	    REGION Niveaumessung
	        // Füllstand Versorgung Frischsäure
	        "Analogwert"(Deaktiviert:=FALSE,
	                                                                                                                                                                                                                                                                                                                                                                                                                                                                                                                                                                                                                                                                                                                                                                                                                                                                                                                                                                                                                                                                                                                                                                                                                                                                                                                                                                                                                                                                                                                                                                                                                                                                                                                                                                                                                                                                                                                                                                                                                                                                                                                                                                                                                                                                                                                                                                                                                                                                                                                                                                                                                                                                                                                                                                                                                                                                                                                                                                                                                                                                                                                                                                                                                                                                                                                                                                                                                                                                                                                                                                                                                                                                                                                                                                                                                                                                                                                                                                                                                                                                                                                                                                                                                                                                                                                                                                                                                                                                                                                                                                                                                                                                                                                                                                                                                                                                                                                                                                                                                                                                                                                                                                                                                                                                                                                                                                                                                                                                                                                                                                                                                                                                                                                                                                                                                                                                                                                                                                                                                                                                                                                                                                                                                                                                                                                                                                                                                                                                                                                                                                                                                                                                                                                                                                                                                                                                                                                                                                                                                                                                                                                                                                                                                                                                                                                                                                                                                                                                                                                                                                                                                                                                                                                                                                                                                                                                                                                                                                                                                                                                                                                                                                                                                                                                                                                                                                                                                                                                                                                                                                                                                                                                                                                                                                                                                                                                                                                                                                                                                                                                                                                                                                                                                                                                                                                                                                                                                                                                                                                                                                                                                                                                                                                                                                                                                                                                                                                                                                                                                                                                                                                                                                                                                                                                                                                                                                                                                                                                                                                                                                                                                                                                                                                                                                                                                                                                                                                                                                                                                                                                                                                                                                                                                                                                                                                                                                                                                                                                                                                                                                                                                                                                                                                                                                                                                                                                                                                                                                                                                                                                                                                                                                                                                                                                                                                                                                                                                                                                                                                                                                                                                                                                                                                                                                                                                                                                                                                                                                                                                                                                                                                                                                                                                                                                                                                                                                                                                                                                                                                                                                                                                                                                                                                                                                                                                                                                                                                                                                                                                                                                                                                                                                                                                                                                                                                                                                                                                                                                                                                                                                                                                                                                                                                                                                                                                                                                                                                                                                                                                                                                                                                                                                                                                                                                                                                                                                                                                                                                                                                                                                                                                                                                                                                                                                                                                                                                                                                                                                                                                                                                                                                                                                                                                                                                                                                                                                                                                                                                                                                                                                                                                                                                                                                                                                                                                                                                                                                                                                                                                                                                                                                                                                                                                                                                                                                                                                                                                                                                                                                                                                                                                                                                                                                                                                                                                                                                                                                                                                                                                                                                                                                                                                                                                                                                                                                                                                                                                                                                                                                                                                                                                                                                                                                                                                                                                                                                                                                                                                                                                                                                                                                                                                                                                                                                                                                                                                                                                                                                                                                                                                                                                                                                                                                                                                                                                                                                                                                                                                                                                                                                                                                                                                                                                                                                                                                                                                                                                                                                                                                                                                                                                                                                                                                                                                                                                                                                                                                                                                                                                                                                                                                                                                                                                                                                                                                                                                                                                                                                                                                                                                                                                                                                                                                                                                                                                                                                                                                                                                                                                                                                                                                                                                                                                                                                                                                                                                                                                                                                                                                                                                                                                                                                                                                                                                                                                                                                                                                                                                                                                                                                                                                                                                                                                                                                                                                                                                                                                                                                                                                                                                                                                                                                                                                                                                                                                                                                                                                                                                                                                                                                                                                                                                                                                                                                                                                                                                                                                                                                                                                                                                                                                                                                                                                                                                                                                                                                                                                                                                                                                                                                                                                                                                                                                                                                                                                                                                                                                                                                                                                                                                                                                                                                                                                                                                                                                                                                                                                                                                                                                                                                                                                                                                                                                                                                                                                                                                                                                                                                                                                                                                                                                                                                                                                                                                                                                                                                                                                                                                                                                                                                                                                                                                                                                                                                                                                                                                                                                                                                                                                                                                                                                                                                                                                                                                                                                                                                                                                                                                                                                                                                                                                                                                                                                                                                                                                                                                                                                                                                                                                                                                                                                                                                                                                                                                                                                                                                                                                                                                                                                                                                                                                                                                                                                                                                                                                                                                                                                                                                                                                                                                                                                                                                                                                                                                                                                                                                                                                                                                                                                                                                                                                                                                                                                                                                                                                                                                                                                                                                                                                                                                                                                                                                                                                                                                                                                                                                                                                                                                                                                                                                                                                                                                                                                                                                                                                                                                                                                                                                                                                                                                                                                                                                                                                                                                                                                                                                                                                                                                                                                                                                                                                                                                                                                                                                                                                                                                                                                                                                                                                                                                                                                                                                                                                                                                                                                                                                                                                                                                                                                                                                                                                                                                                                                                                                                                                                                                                                                                                                                                                                                                                                                                                                                                                                                                                                                                                                                                                                                                                                                                                                                                                                                                                                                                                                                                                                                                                                                                                                                                                                                                                                                                                                                                                                                                                                                                                                                                                                                                                                                                                                                                                                                                                                                                                                                                                                                                                                                                                                                                                                                                                                                                                                                                                                                                                                                                                                                                                                                                                                                                                                                                                                                                                                                                                                                                                                                                                                                                                                                                                                                                                                                                                                                                                                                                                                                                                                                                                                                                                                                                                                                                                                                                                                                                                                                                                                                                                                                                                                                                                                                                                                                                                                                                                                                                                                                                                                                                                                                                                                                                                                                                                                                                                                                                                                                                                                                                                                                                                                                                                                                                                                                                                                                                                                                                                                                                                                                                                                                                                                                                                                                                                                                                                                                                                                                                                                                                                                                                                                                                                                                                                                                                                                                                                                                                                                                                                                                                                                                                                                                                                                                                                                                                                                                                                                                                                                                                                                                                                                                                                                                                                                                                                                                                                                                                                                                                                                                                                                                                                                                                                                                                                                                                                                                                                                                                                                                                                                                                                                                                                                                                                                                                                                                                                                                                                                                                                                                                                                                                                                                                                                                                                                                                                                                                                                                                                                                                                                                                                                                                                                                                                                                                                                                                                                                                                                                                                                                                                                                                                                                                                                                                                                                                                                                                                                                                                                                                                                                                                                                                                                                                                                                                                                                                                                                                                                                                                                                                                                                                                                                                                                                                                                                                                                                                                                                                                                                                                                                                                                                                                                                                                                                                                                                                                                                                                                                                                                                                                                                                                                                                                                                                                                                                                                                                                                                                                                                                                                                                                                                                                                                                                                                                                                                                                                                                                                                                                                                                                                                                                                                                                                                                                                                                                                                                                                                                                                                                                                                                                                                                                                                                                                                                                                                                                                                                                                                                                                                                                                                                                                                                                                                                                                                                                                                                                                                                                                                                                                                                                                                                                                                                                                                                                                                                                                                                                                                                                                                                                                                                                                                                                                                                                                                                                                                                                                                                                                                                                                                                                                                                                                                                                                                                                                                                                                                                                                                                                                                                                                                                                                                                                                                                                                                                                                                                                                                                                                                                                                                                                                                                                                                                                                                                                                                                                                                                                                                                                                                                                                                                                                                                                                                                                                                                                                                                                                                                                                                                                                                                                                                                                                                                                                                                                                                                                                                                                                                                                                                                                                                                                                                                                                                                                                                                                                                                                                                                                                                                                                                                                                                                                                                                                                                                                                                                                                                                                                                                                                                                                                                                                                                                                                                                                                                                                                                                                                                                                                                                                                                                                                                                                                                                                                                                                                                                                                                                                                                                                                                                                                                                                                                                                                                                                                                                                                                                                                                                                                                                                                                                                                                                                                                                                                                                                                                                                                                                                                                                                                                                                                                                                                                                                                                                                                                                                                                                                                                                                                                                                                                                                                                                                                                                                                                                                                                                                                                                                                                                                                                                                                                                                                                                                                                                                                                                                                                                                                                                                                                                                                                                                                                                                                                                                                                                                                                                                                                                                                                                                                                                                                                                                                                                                                                                                                                                                                                                                                                                                                                                                                                                                                                                                                                                                                                                                                                                                                                                                                                                                                                                                                                                                                                                                                                                                                                                                                                                                                                                                                                                                                                                                                                                                                                                                                                                                                                                                                                                                                                                                                                                                                                                                                                                                                                                                                                                                                                                                                                                                                                                                                                                                                                                                                                                                                                                                                                                                                                                                                                                                                                                                                                                                                                                                                                                                                                                                                                                                                                                                                                                                                                                                                                                                                                                                                                                                                                                                                                                                                                                                                                                                                                                                                                                                                                                                                                                                                                                                                                                                                                                                                                                                                                                                                                                                                                                                                                                                                                                                                                                                                                                                                                                                                                                                                                                                                                                                                                                                                                                                                                                                                                                                                                                                                                                                                                                                                                                                                                                                                                                                                                                                                                                                                                                                                                                                                                                                                                                                                                                                                                                                                                                                                                                                                                                                                                                                                                                                                                                                                                                                                                                                                                                                                                                                                                                                                                                                                                                                                                                                                                                                                                                                                                                                                                                                                                                                                                                                                                                                                                                                                                                                                                                                                                                                                                                                                                                                                                                                                                                                                                                                                                                                                                                                                                                                                                                                                                                                                                                                                                                                                                                                                                                                                                                                                                                                                                                                                                                                                                                                                                                                                                                                                                                                                                                                                                                                                                                                                                                                                                                                                                                                                                                                                                                                                                                                                                                                                                                                                                                                                                                                                                                                                                                                                                                                                                                                                                                                                                                                                                                                                                                                                                                                                                                                                                                                                                                                                                                                                                                                                                                                                                                                                                                                                                                                                                                                                                                                                                                                                                                                                                                                                                                                                                                                                                      EW := "EW_Niv_GP01.BL30",
	                     Messbereich_Min := "Analogwerte"."Niv_GP01.BL30".MB_min,
	                     Messbereich_Max := "Analogwerte"."Niv_GP01.BL30".MB_max,
	                     UG_Alarm := "Analogwerte"."Niv_GP01.BL30".UG_Alarm,
	                     OG_Alarm := "Analogwerte"."Niv_GP01.BL30".OG_Alarm,
	                     GF := "Analogwerte"."Niv_GP01.BL30".GF,
	                     Al_Drahtbruch => "Analogwerte"."Niv_GP01.BL30".Drahtbruch,
	                     Al_MW_ausserhalb => "Analogwerte"."Niv_GP01.BL30".ungueltig,
	                     Messwert := "Panel".IW."Niv_GP01.BL30");
	        // Füllstand Entsorgung Altsäure
	        "Analogwert"(Deaktiviert:=FALSE,
	                        EW := "EW_Niv_GP02.BL31",
	                     Messbereich_Min := "Analogwerte"."Niv_GP02.BL31".MB_min,
	                     Messbereich_Max := "Analogwerte"."Niv_GP02.BL31".MB_max,
	                     UG_Alarm := "Analogwerte"."Niv_GP02.BL31".UG_Alarm,
	                     OG_Alarm := "Analogwerte"."Niv_GP02.BL31".OG_Alarm,
	                     GF := "Analogwerte"."Niv_GP02.BL31".GF,
	                     Al_Drahtbruch => "Analogwerte"."Niv_GP02.BL31".Drahtbruch,
	                     Al_MW_ausserhalb => "Analogwerte"."Niv_GP02.BL31".ungueltig,
	                     Messwert := "Panel".IW."Niv_GP02.BL31");
	     END_REGION
	// pH-Messung
	     "Analogwert"(Deaktiviert:=FALSE,
	             EW := "EW_LW_BE",
	             Messbereich_Min := "Analogwerte".pH_WR01.MB_min,
	             Messbereich_Max := "Analogwerte".pH_WR01.MB_max,
	             UG_Alarm := "Analogwerte".pH_WR01.UG_Alarm,
	             OG_Alarm := "Analogwerte".pH_WR01.OG_Alarm,
	             GF := "Analogwerte".pH_WR01.GF,
	             Al_Drahtbruch => "Analogwerte".pH_WR01.Drahtbruch,
	             Al_MW_ausserhalb => "Analogwerte".pH_WR01.ungueltig,
	             Messwert := "Panel".IW."pH_BE");
	END_IF;
	
	REGION Manipulator
	    IF "Imp_10Hz" THEN // 8x Wägezelle, 2x Last
	        "Analogwert"(Deaktiviert:=FALSE,
	                     EW := "EW_WZ_links_1",
	                     Messbereich_Min := "Analogwerte".WZ_1_1.MB_min,
	                     Messbereich_Max := "Analogwerte".WZ_1_1.MB_max,
	                     UG_Alarm := "Analogwerte".WZ_1_1.UG_Alarm,
	                     OG_Alarm := "Analogwerte".WZ_1_1.OG_Alarm,
	                     GF := "Analogwerte".WZ_1_1.GF,
	                     Al_Drahtbruch => "Analogwerte".WZ_1_1.Drahtbruch,
	                     Al_MW_ausserhalb => "Analogwerte".WZ_1_1.ungueltig,
	                     Messwert := "DI_FW_1".HELP.WZ_links_1);
	        
	        "Analogwert"(Deaktiviert:=FALSE,
	                     EW := "EW_WZ_links_2",
	                     Messbereich_Min := "Analogwerte".WZ_1_2.MB_min,
	                     Messbereich_Max := "Analogwerte".WZ_1_2.MB_max,
	                     UG_Alarm := "Analogwerte".WZ_1_2.UG_Alarm,
	                     OG_Alarm := "Analogwerte".WZ_1_2.OG_Alarm,
	                     GF := "Analogwerte".WZ_1_2.GF,
	                     Al_Drahtbruch => "Analogwerte".WZ_1_2.Drahtbruch,
	                     Al_MW_ausserhalb => "Analogwerte".WZ_1_2.ungueltig,
	                     Messwert := "DI_FW_1".HELP.WZ_links_2);
	        
	        "Analogwert"(Deaktiviert:=FALSE,
	                     EW := "EW_WZ_links_3",
	                     Messbereich_Min := "Analogwerte".WZ_1_3.MB_min,
	                     Messbereich_Max := "Analogwerte".WZ_1_3.MB_max,
	                     UG_Alarm := "Analogwerte".WZ_1_3.UG_Alarm,
	                     OG_Alarm := "Analogwerte".WZ_1_3.OG_Alarm,
	                     GF := "Analogwerte".WZ_1_3.GF,
	                     Al_Drahtbruch => "Analogwerte".WZ_1_3.Drahtbruch,
	                     Al_MW_ausserhalb => "Analogwerte".WZ_1_3.ungueltig,
	                     Messwert := "DI_FW_1".HELP.WZ_links_3);
	        
	        "Analogwert"(Deaktiviert:=FALSE,
	                    EW := "EW_WZ_links_4",
	                     Messbereich_Min := "Analogwerte".WZ_1_4.MB_min,
	                     Messbereich_Max := "Analogwerte".WZ_1_4.MB_max,
	                     UG_Alarm := "Analogwerte".WZ_1_4.UG_Alarm,
	                     OG_Alarm := "Analogwerte".WZ_1_4.OG_Alarm,
	                     GF := "Analogwerte".WZ_1_4.GF,
	                     Al_Drahtbruch => "Analogwerte".WZ_1_4.Drahtbruch,
	                     Al_MW_ausserhalb => "Analogwerte".WZ_1_4.ungueltig,
	                     Messwert := "DI_FW_1".HELP.WZ_links_4);
	        
	        "Analogwert"(Deaktiviert:=FALSE,
	                     EW := "EW_WZ_rechts_1",
	                     Messbereich_Min := "Analogwerte".WZ_2_1.MB_min,
	                     Messbereich_Max := "Analogwerte".WZ_2_1.MB_max,
	                     UG_Alarm := "Analogwerte".WZ_2_1.UG_Alarm,
	                     OG_Alarm := "Analogwerte".WZ_2_1.OG_Alarm,
	                     GF := "Analogwerte".WZ_2_1.GF,
	                     Al_Drahtbruch => "Analogwerte".WZ_2_1.Drahtbruch,
	                     Al_MW_ausserhalb => "Analogwerte".WZ_2_1.ungueltig,
	                     Messwert := "DI_FW_1".HELP.WZ_rechts_1);
	        
	        "Analogwert"(Deaktiviert := FALSE,
	                     EW := "EW_WZ_rechts_2",
	                     Messbereich_Min := "Analogwerte".WZ_2_2.MB_min,
	                     Messbereich_Max := "Analogwerte".WZ_2_2.MB_max,
	                     UG_Alarm := "Analogwerte".WZ_2_2.UG_Alarm,
	                     OG_Alarm := "Analogwerte".WZ_2_2.OG_Alarm,
	                     GF := "Analogwerte".WZ_2_2.GF,
	                     Al_Drahtbruch => "Analogwerte".WZ_2_2.Drahtbruch,
	                     Al_MW_ausserhalb => "Analogwerte".WZ_2_2.ungueltig,
	                     Messwert := "DI_FW_1".HELP.WZ_rechts_2);
	        
	        "Analogwert"(Deaktiviert := FALSE,
	                     EW := "EW_WZ_rechts_3",
	                     Messbereich_Min := "Analogwerte".WZ_2_3.MB_min,
	                     Messbereich_Max := "Analogwerte".WZ_2_3.MB_max,
	                     UG_Alarm := "Analogwerte".WZ_2_3.UG_Alarm,
	                     OG_Alarm := "Analogwerte".WZ_2_3.OG_Alarm,
	                     GF := "Analogwerte".WZ_2_3.GF,
	                     Al_Drahtbruch => "Analogwerte".WZ_2_3.Drahtbruch,
	                     Al_MW_ausserhalb => "Analogwerte".WZ_2_3.ungueltig,
	                     Messwert := "DI_FW_1".HELP.WZ_rechts_3);
	        
	        "Analogwert"(Deaktiviert := FALSE,
	                     EW := "EW_WZ_rechts_4",
	                     Messbereich_Min := "Analogwerte".WZ_2_4.MB_min,
	                     Messbereich_Max := "Analogwerte".WZ_2_4.MB_max,
	                     UG_Alarm := "Analogwerte".WZ_2_4.UG_Alarm,
	                     OG_Alarm := "Analogwerte".WZ_2_4.OG_Alarm,
	                     GF := "Analogwerte".WZ_2_4.GF,
	                     Al_Drahtbruch => "Analogwerte".WZ_2_4.Drahtbruch,
	                     Al_MW_ausserhalb => "Analogwerte".WZ_2_4.ungueltig,
	                     Messwert := "DI_FW_1".HELP.WZ_rechts_4);
	        
	        "Analogwert"(Deaktiviert := FALSE,
	                     EW := "EW_Last_links",
	                     Messbereich_Min := "Analogwerte".Last_1.MB_min,
	                     Messbereich_Max := "Analogwerte".Last_1.MB_max,
	                     UG_Alarm := "Analogwerte".Last_1.UG_Alarm,
	                     OG_Alarm := "Analogwerte".Last_1.OG_Alarm,
	                     GF := "Analogwerte".Last_1.GF,
	                     Al_Drahtbruch => "Analogwerte".Last_1.Drahtbruch,
	                     Al_MW_ausserhalb => "Analogwerte".Last_1.ungueltig,
	                     Messwert := "DI_FW_1".HELP.Last_1);
	        
	        "Analogwert"(Deaktiviert:=FALSE,
	                     EW := "EW_Last_rechts",
	                     Messbereich_Min := "Analogwerte".Last_2.MB_min,
	                     Messbereich_Max := "Analogwerte".Last_2.MB_max,
	                     UG_Alarm := "Analogwerte".Last_2.UG_Alarm,
	                     OG_Alarm := "Analogwerte".Last_2.OG_Alarm,
	                     GF := "Analogwerte".Last_2.GF,
	                     Al_Drahtbruch => "Analogwerte".Last_2.Drahtbruch,
	                     Al_MW_ausserhalb => "Analogwerte".Last_2.ungueltig,
	                     Messwert := "DI_FW_1".HELP.Last_2);
	    END_IF;
	
	END_REGION
	
END_FUNCTION

FUNCTION "Analogwert" : Void
{ S7_Optimized_Access := 'TRUE' }
VERSION : 0.1
   VAR_INPUT 
      Deaktiviert : Bool;
      EW : Int;
      Messbereich_Min : Real;
      Messbereich_Max : Real;
      UG_Alarm : Real;
      OG_Alarm : Real;
      GF : Real;
   END_VAR

   VAR_OUTPUT 
      Al_Drahtbruch : Bool;
      Al_MW_ausserhalb : Bool;
   END_VAR

   VAR_IN_OUT 
      Messwert : Real;
   END_VAR

   VAR_TEMP 
      akt_Messwert : Real;
      Messbereich : Real;
      Eingangswert : Real;
   END_VAR

   VAR CONSTANT 
      Drahtbruchkennung : Int := 16#7FFF;
      Defekt : Int := 16#8000;
      EW_min : Real;
      EW_max : Real := 27648.0;   // SIEMENS-Baugruppe (0x6C00)
   END_VAR


BEGIN
	IF #Deaktiviert THEN //20.01.22
	    #Al_Drahtbruch := FALSE;
	    #Al_MW_ausserhalb := false;
	    #Messwert := 0.0;
	    
	ELSIF (#EW = #Drahtbruchkennung) OR (#EW = #Defekt) THEN
	    #Al_Drahtbruch := TRUE;
	    #Al_MW_ausserhalb := false;
	    #Messwert := 0.0;
	ELSE
	    #Al_Drahtbruch := FALSE;
	    #Messbereich := (#EW_max - #EW_min);
	    #Eingangswert := DINT_TO_REAL(INT_TO_DINT(#EW));
	    
	    #akt_Messwert := ((#Eingangswert - #EW_min) * #Messbereich_Max / #Messbereich) + ((#EW_max - #Eingangswert) * #Messbereich_Min / #Messbereich);
	      
	    IF (#GF <= 0.0) OR #GF >= 1.0 THEN
	        #Messwert := #akt_Messwert;
	    ELSE
	         #Messwert := (#akt_Messwert * #GF) + ((1.0 - #GF) * #Messwert);
	     END_IF;
	     #Al_MW_ausserhalb := (#Messwert < #UG_Alarm) OR (#Messwert > #OG_Alarm);
	    
	END_IF;
	
END_FUNCTION

FUNCTION "BA_WXL" : Void   // FC4, STL
{ S7_Optimized_Access := 'FALSE' }
AUTHOR : MS
// stored: AutoNumber false
   VAR_TEMP
      Evnt_Nbr : Byte;
   END_VAR
   VAR CONSTANT
      Not_Halt : USInt;
      Tipp : USInt := 1;
      Hand : USInt := 2;
      Automat_Aus : USInt := 3;
      Automat_Ein : USInt := 4;
   END_VAR
BEGIN

NETWORK
TITLE = Not-Aus ist betätigt
      A     "DB_ANLAGE".config.Anl_getaktet;
      =     "DB_Panel_OVERVIEW".SPS_getaktet;

      A     "DB_ANLAGE".IN.S_Not_Aus;
      JC    off;

//Automatikbetrieb
      A     "DB_ANLAGE".BA.Not_Aus;
      R     "DB_ANLAGE".BA.Not_Aus;
      R     "DB_ANLAGE".BA.Tippbetrieb;
      R     "DB_ANLAGE".BA.Handbetrieb;
      R     "DB_ANLAGE".BA.Automat_ein;
      S     "DB_ANLAGE".BA.Automat_aus;

      A     "DB_ANLAGE".IN.Automat_ein;
      FP    "DB_ANLAGE".BA.FP_Automat_ein;
      R     "DB_ANLAGE".BA.Not_Aus;
      R     "DB_ANLAGE".BA.Tippbetrieb;
      R     "DB_ANLAGE".BA.Handbetrieb;
      S     "DB_ANLAGE".BA.Automat_ein;
      R     "DB_ANLAGE".BA.Automat_aus;

      A     "DB_ANLAGE".IN.Automat_aus;
      R     "DB_ANLAGE".BA.Not_Aus;
      R     "DB_ANLAGE".BA.Tippbetrieb;
      R     "DB_ANLAGE".BA.Handbetrieb;
      R     "DB_ANLAGE".BA.Automat_ein;
      S     "DB_ANLAGE".BA.Automat_aus;

      A     "DB_ANLAGE".BA.Automat_ein;
      O     "DI_FW_MANAGER".Auto.Anlage;
      O     "DB_ANLAGE".IN.Lamp_Test;
      =     "DB_ANLAGE".OUT.MD_Auto;

//Handbetrieb
      A     "DB_ANLAGE".IN.BA_Hand;
      R     "DB_ANLAGE".BA.Not_Aus;
      R     "DB_ANLAGE".BA.Tippbetrieb;
      S     "DB_ANLAGE".BA.Handbetrieb;
      R     "DB_ANLAGE".BA.Automat_ein;
      R     "DB_ANLAGE".BA.Automat_aus;

//Einrichten
      A     "DB_ANLAGE".IN.BA_Tipp;
      R     "DB_ANLAGE".BA.Not_Aus;
      S     "DB_ANLAGE".BA.Tippbetrieb;
      R     "DB_ANLAGE".BA.Handbetrieb;
      R     "DB_ANLAGE".BA.Automat_ein;
      R     "DB_ANLAGE".BA.Automat_aus;

//Auto-Stop
      A     "DB_ANLAGE".BA.Automat_aus;
      R     "DB_ANLAGE".BA.Not_Aus;
      R     "DB_ANLAGE".BA.Tippbetrieb;
      R     "DB_ANLAGE".BA.Handbetrieb;
      R     "DB_ANLAGE".BA.Automat_ein;

      L     #Automat_Ein;
      A     "DB_ANLAGE".BA.Automat_ein;
      JC    A_BA;
      L     #Automat_Aus;
      A     "DB_ANLAGE".BA.Automat_aus;
      JC    A_BA;
      L     #Hand;
      A     "DB_ANLAGE".BA.Handbetrieb;
      JC    A_BA;
      L     #Tipp;
      A     "DB_ANLAGE".BA.Tippbetrieb;
      JC    A_BA;
      L     #Not_Halt;
A_BA: T     "Panel".Betriebsart.Anzeige;
      JU    ende;

//alles aus
off:  R     "DB_ANLAGE".BA.free0;
      R     "DB_ANLAGE".BA.free1;
      R     "DB_ANLAGE".BA.Tippbetrieb;
      R     "DB_ANLAGE".BA.Handbetrieb;
      R     "DB_ANLAGE".BA.Automat_ein;
      R     "DB_ANLAGE".BA.Automat_aus;
      S     "DB_ANLAGE".BA.Not_Aus;
      L     #Not_Halt;
      T     "Panel".Betriebsart.Anzeige;

ende: OPN   "DB_ANLAGE";
      L     %DBW0;  //Betriebsart SPS
      OPN   "DB_Panel_OVERVIEW";
      T     %DBW0;  //Betriebsart Visualisierung
      BE;
END_FUNCTION

FUNCTION "FC_Optimierung" : Void   // FC170, STL
{ S7_Optimized_Access := 'TRUE' }
// stored: AutoNumber false
   VAR_TEMP
      Count : Int;
      WT_DB : Int;
      Cmd : Int;
      Restzeit : DInt;
      Umsetzzeit : DInt;
      Restzeit_Kurz_Links : DInt;
      Restzeit_Kurz_Rechts : DInt;
      Restzeit_Lang : DInt;
      Restzeit_Gross_Links : DInt;
      Restzeit_Gross_Rechts : DInt;
      Belegt : Array[1..18] of Bool;
      Lang : Array[1..6] of Bool;
   END_VAR
BEGIN

NETWORK
TITLE = Restzeiten ermitteln
      AN    "Imp_0.5Hz";
      BEC;

      L     180;
      T     #Umsetzzeit;

//CM01
//links mitte Großoptik
      CALL  "FC_Optimierung_Pos"
      ( Pos        := 3,
        Umsetzzeit := #Umsetzzeit,
        Belegt     := #Belegt[3],
        Restzeit   := "DB_Optimierung_HCA".Restzeit[3]
      );

      L     0;
      T     "DB_Optimierung_HCA".Restzeit[1];
      T     "DB_Optimierung_HCA".Restzeit[5];

      SET;
      R     #Lang[1];
      R     #Lang[2];
      R     #Belegt[1];
      R     #Belegt[5];

      A     #Belegt[3];
      JC    cR1M;

//links rückwärts
cL1R: CALL  "FC_Optimierung_Pos"
      ( Pos        := 1,
        Umsetzzeit := #Umsetzzeit,
        Belegt     := #Belegt[1],
        Restzeit   := "DB_Optimierung_HCA".Restzeit[1]
      );

      L     "DB_POS".POS[1].next_WT;
      L     "DB_POS".POS[2].next_WT;
      ==I;
      A     #Belegt[1];
      =     #Lang[1];

//links vorwärts
cL1V: CALL  "FC_Optimierung_Pos"
      ( Pos        := 5,
        Umsetzzeit := #Umsetzzeit,
        Belegt     := #Belegt[5],
        Restzeit   := "DB_Optimierung_HCA".Restzeit[5]
      );

      L     "DB_POS".POS[5].next_WT;
      L     "DB_POS".POS[6].next_WT;
      ==I;
      A     #Belegt[5];
      =     #Lang[2];

//rechts mitte Großoptik
cR1M: CALL  "FC_Optimierung_Pos"
      ( Pos        := 4,
        Umsetzzeit := #Umsetzzeit,
        Belegt     := #Belegt[4],
        Restzeit   := "DB_Optimierung_HCA".Restzeit[4]
      );

      L     0;
      T     "DB_Optimierung_HCA".Restzeit[2];
      T     "DB_Optimierung_HCA".Restzeit[6];

      SET;
      R     #Belegt[2];
      R     #Belegt[6];

      A     #Belegt[4];
      JC    cL2M;

//rechts rückwärts
cR1R: A     #Belegt[1];
      =     #Belegt[2];

      L     "DB_Optimierung_HCA".Restzeit[1];
      T     "DB_Optimierung_HCA".Restzeit[2];

      A     #Lang[1];
      JC    cR1V;

      CALL  "FC_Optimierung_Pos"
      ( Pos        := 2,
        Umsetzzeit := #Umsetzzeit,
        Belegt     := #Belegt[2],
        Restzeit   := "DB_Optimierung_HCA".Restzeit[2]
      );

//rechts vorwärts
cR1V: A     #Belegt[5];
      =     #Belegt[6];

      L     "DB_Optimierung_HCA".Restzeit[5];
      T     "DB_Optimierung_HCA".Restzeit[6];

      A     #Lang[2];
      JC    cL2M;

      CALL  "FC_Optimierung_Pos"
      ( Pos        := 6,
        Umsetzzeit := #Umsetzzeit,
        Belegt     := #Belegt[6],
        Restzeit   := "DB_Optimierung_HCA".Restzeit[6]
      );

//CM02
//links mitte
cL2M: CALL  "FC_Optimierung_Pos"
      ( Pos        := 15,
        Umsetzzeit := #Umsetzzeit,
        Belegt     := #Belegt[15],
        Restzeit   := "DB_Optimierung_HCA".Restzeit[15]
      );

      L     0;
      T     "DB_Optimierung_HCA".Restzeit[13];
      T     "DB_Optimierung_HCA".Restzeit[17];

      SET;
      R     #Lang[5];
      R     #Lang[6];
      R     #Belegt[13];
      R     #Belegt[17];

      A     #Belegt[15];
      JC    cR2M;

//links rüclwärts
cL2R: CALL  "FC_Optimierung_Pos"
      ( Pos        := 13,
        Umsetzzeit := #Umsetzzeit,
        Belegt     := #Belegt[13],
        Restzeit   := "DB_Optimierung_HCA".Restzeit[13]
      );

      L     "DB_POS".POS[13].next_WT;
      L     "DB_POS".POS[14].next_WT;
      ==I;
      A     #Belegt[13];
      =     #Lang[5];

//links vorwärts
cL2V: CALL  "FC_Optimierung_Pos"
      ( Pos        := 17,
        Umsetzzeit := #Umsetzzeit,
        Belegt     := #Belegt[17],
        Restzeit   := "DB_Optimierung_HCA".Restzeit[17]
      );

      L     "DB_POS".POS[17].next_WT;
      L     "DB_POS".POS[18].next_WT;
      ==I;
      A     #Belegt[17];
      =     #Lang[6];

//rechts mitte
cR2M: CALL  "FC_Optimierung_Pos"
      ( Pos        := 16,
        Umsetzzeit := #Umsetzzeit,
        Belegt     := #Belegt[16],
        Restzeit   := "DB_Optimierung_HCA".Restzeit[16]
      );

      L     0;
      T     "DB_Optimierung_HCA".Restzeit[14];
      T     "DB_Optimierung_HCA".Restzeit[18];

      SET;
      R     #Belegt[14];
      R     #Belegt[18];

      A     #Belegt[16];
      JC    cL3M;

//rechts rückwärts
cR2R: A     #Belegt[13];
      =     #Belegt[14];

      L     "DB_Optimierung_HCA".Restzeit[13];
      T     "DB_Optimierung_HCA".Restzeit[14];

      A     #Lang[5];
      JC    cR2V;

      CALL  "FC_Optimierung_Pos"
      ( Pos        := 14,
        Umsetzzeit := #Umsetzzeit,
        Belegt     := #Belegt[14],
        Restzeit   := "DB_Optimierung_HCA".Restzeit[14]
      );

//rechts vorwärts
cR2V: A     #Belegt[17];
      =     #Belegt[18];

      L     "DB_Optimierung_HCA".Restzeit[17];
      T     "DB_Optimierung_HCA".Restzeit[18];

      A     #Lang[6];
      JC    cL3M;

      CALL  "FC_Optimierung_Pos"
      ( Pos        := 18,
        Umsetzzeit := #Umsetzzeit,
        Belegt     := #Belegt[18],
        Restzeit   := "DB_Optimierung_HCA".Restzeit[18]
      );

//CM03
//links mitte
cL3M: CALL  "FC_Optimierung_Pos"
      ( Pos        := 9,
        Umsetzzeit := #Umsetzzeit,
        Belegt     := #Belegt[9],
        Restzeit   := "DB_Optimierung_HCA".Restzeit[9]
      );

      L     0;
      T     "DB_Optimierung_HCA".Restzeit[7];
      T     "DB_Optimierung_HCA".Restzeit[11];

      SET;
      R     #Lang[3];
      R     #Lang[4];
      R     #Belegt[7];
      R     #Belegt[11];

      AN    #Belegt[9];
      JC    cL3R;

      A     #Belegt[1];
      O     #Belegt[3];
      O     #Belegt[5];
      JC    cL3M2;
      S     #Belegt[3];

      L     "DB_Optimierung_HCA".Restzeit[9];
      T     "DB_Optimierung_HCA".Restzeit[3];
      JU    cR3M;

cL3M2:A     #Belegt[13];
      O     #Belegt[15];
      O     #Belegt[17];
      JC    cR3M;
      S     #Belegt[15];

      L     "DB_Optimierung_HCA".Restzeit[9];
      T     "DB_Optimierung_HCA".Restzeit[15];
      JU    cR3M;

cL3R: CALL  "FC_Optimierung_Pos"
      ( Pos        := 7,
        Umsetzzeit := #Umsetzzeit,
        Belegt     := #Belegt[7],
        Restzeit   := "DB_Optimierung_HCA".Restzeit[7]
      );

      L     "DB_POS".POS[7].next_WT;
      L     "DB_POS".POS[8].next_WT;
      ==I;
      A     #Belegt[7];
      =     #Lang[3];

      AN    #Belegt[7];
      JC    cL3V;

      AN    #Belegt[2];
      AN    #Belegt[4];
      ON    #Lang[3];
      AN    #Belegt[1];
      AN    #Belegt[3];
      JC    cL3R_1R;

      AN    #Belegt[6];
      AN    #Belegt[4];
      ON    #Lang[3];
      AN    #Belegt[5];
      AN    #Belegt[3];
      JC    cL3R_1V;

      AN    #Belegt[14];
      AN    #Belegt[16];
      ON    #Lang[3];
      AN    #Belegt[13];
      AN    #Belegt[15];
      JC    cL3R_2R;

      AN    #Belegt[18];
      AN    #Belegt[16];
      ON    #Lang[3];
      AN    #Belegt[17];
      AN    #Belegt[15];
      JC    cL3R_2V;

      JU    cL3V;

cL3R_1R:SET;
      S     #Belegt[1];
      L     "DB_Optimierung_HCA".Restzeit[7];
      T     "DB_Optimierung_HCA".Restzeit[1];

      AN    #Lang[3];
      JC    cL3V;
      S     #Belegt[2];
      L     "DB_Optimierung_HCA".Restzeit[7];
      T     "DB_Optimierung_HCA".Restzeit[2];
      JU    cL3V;

cL3R_1V:SET;
      S     #Belegt[5];
      L     "DB_Optimierung_HCA".Restzeit[7];
      T     "DB_Optimierung_HCA".Restzeit[5];

      AN    #Lang[3];
      JC    cL3V;
      S     #Belegt[6];
      L     "DB_Optimierung_HCA".Restzeit[7];
      T     "DB_Optimierung_HCA".Restzeit[6];
      JU    cL3V;

cL3R_2R:SET;
      S     #Belegt[13];
      L     "DB_Optimierung_HCA".Restzeit[7];
      T     "DB_Optimierung_HCA".Restzeit[13];

      AN    #Lang[3];
      JC    cL3V;
      S     #Belegt[14];
      L     "DB_Optimierung_HCA".Restzeit[7];
      T     "DB_Optimierung_HCA".Restzeit[14];
      JU    cL3V;

cL3R_2V:SET;
      S     #Belegt[17];
      L     "DB_Optimierung_HCA".Restzeit[7];
      T     "DB_Optimierung_HCA".Restzeit[17];

      AN    #Lang[3];
      JC    cL3V;
      S     #Belegt[18];
      L     "DB_Optimierung_HCA".Restzeit[7];
      T     "DB_Optimierung_HCA".Restzeit[18];
      JU    cL3V;

cL3V: CALL  "FC_Optimierung_Pos"
      ( Pos        := 11,
        Umsetzzeit := #Umsetzzeit,
        Belegt     := #Belegt[11],
        Restzeit   := "DB_Optimierung_HCA".Restzeit[11]
      );

      L     "DB_POS".POS[11].next_WT;
      L     "DB_POS".POS[12].next_WT;
      ==I;
      A     #Belegt[11];
      =     #Lang[4];

      AN    #Belegt[11];
      JC    cR3M;

      AN    #Belegt[2];
      AN    #Belegt[4];
      ON    #Lang[4];
      AN    #Belegt[1];
      AN    #Belegt[3];
      JC    cL3V_1R;

      AN    #Belegt[6];
      AN    #Belegt[4];
      ON    #Lang[4];
      AN    #Belegt[5];
      AN    #Belegt[3];
      JC    cL3V_1V;

      AN    #Belegt[14];
      AN    #Belegt[16];
      ON    #Lang[4];
      AN    #Belegt[13];
      AN    #Belegt[15];
      JC    cL3V_2R;

      AN    #Belegt[18];
      AN    #Belegt[16];
      ON    #Lang[4];
      AN    #Belegt[17];
      AN    #Belegt[15];
      JC    cL3V_2V;

      JU    cR3M;

cL3V_1R:SET;
      S     #Belegt[1];
      L     "DB_Optimierung_HCA".Restzeit[11];
      T     "DB_Optimierung_HCA".Restzeit[1];

      AN    #Lang[4];
      JC    cR3M;
      S     #Belegt[2];
      L     "DB_Optimierung_HCA".Restzeit[11];
      T     "DB_Optimierung_HCA".Restzeit[2];
      JU    cR3M;

cL3V_1V:SET;
      S     #Belegt[5];
      L     "DB_Optimierung_HCA".Restzeit[11];
      T     "DB_Optimierung_HCA".Restzeit[5];

      AN    #Lang[4];
      JC    cR3M;
      S     #Belegt[6];
      L     "DB_Optimierung_HCA".Restzeit[11];
      T     "DB_Optimierung_HCA".Restzeit[6];
      JU    cR3M;

cL3V_2R:SET;
      S     #Belegt[13];
      L     "DB_Optimierung_HCA".Restzeit[11];
      T     "DB_Optimierung_HCA".Restzeit[13];

      AN    #Lang[4];
      JC    cR3M;
      S     #Belegt[14];
      L     "DB_Optimierung_HCA".Restzeit[11];
      T     "DB_Optimierung_HCA".Restzeit[14];
      JU    cR3M;

cL3V_2V:SET;
      S     #Belegt[17];
      L     "DB_Optimierung_HCA".Restzeit[11];
      T     "DB_Optimierung_HCA".Restzeit[17];

      AN    #Lang[4];
      JC    cR3M;
      S     #Belegt[18];
      L     "DB_Optimierung_HCA".Restzeit[11];
      T     "DB_Optimierung_HCA".Restzeit[18];
      JU    cR3M;

//rechts mitte
cR3M: CALL  "FC_Optimierung_Pos"
      ( Pos        := 10,
        Umsetzzeit := #Umsetzzeit,
        Belegt     := #Belegt[10],
        Restzeit   := "DB_Optimierung_HCA".Restzeit[10]
      );

      L     0;
      T     "DB_Optimierung_HCA".Restzeit[8];
      T     "DB_Optimierung_HCA".Restzeit[12];

      SET;
      R     #Belegt[8];
      R     #Belegt[12];

      AN    #Belegt[10];
      JC    cR3R;

      A     #Belegt[2];
      O     #Belegt[4];
      O     #Belegt[6];
      JC    cR3M2;
      S     #Belegt[4];

      L     "DB_Optimierung_HCA".Restzeit[10];
      T     "DB_Optimierung_HCA".Restzeit[4];
      JU    cEnd;

cR3M2:A     #Belegt[14];
      O     #Belegt[16];
      O     #Belegt[18];
      JC    cEnd;
      S     #Belegt[16];

      L     "DB_Optimierung_HCA".Restzeit[10];
      T     "DB_Optimierung_HCA".Restzeit[16];
      JU    cEnd;

cR3R: A     #Belegt[7];
      A     #Lang[3];
      JC    cR3V;

      CALL  "FC_Optimierung_Pos"
      ( Pos        := 8,
        Umsetzzeit := #Umsetzzeit,
        Belegt     := #Belegt[8],
        Restzeit   := "DB_Optimierung_HCA".Restzeit[8]
      );

      AN    #Belegt[8];
      JC    cR3V;

      AN    #Belegt[2];
      AN    #Belegt[4];
      JC    cR3R_1R;

      AN    #Belegt[6];
      AN    #Belegt[4];
      JC    cR3R_1V;

      AN    #Belegt[14];
      AN    #Belegt[16];
      JC    cR3R_2R;

      AN    #Belegt[18];
      AN    #Belegt[16];
      JC    cR3R_2V;

      JU    cR3V;

cR3R_1R:SET;
      S     #Belegt[2];
      L     "DB_Optimierung_HCA".Restzeit[8];
      T     "DB_Optimierung_HCA".Restzeit[2];
      JU    cR3V;

cR3R_1V:SET;
      S     #Belegt[6];
      L     "DB_Optimierung_HCA".Restzeit[8];
      T     "DB_Optimierung_HCA".Restzeit[6];
      JU    cR3V;

cR3R_2R:SET;
      S     #Belegt[14];
      L     "DB_Optimierung_HCA".Restzeit[8];
      T     "DB_Optimierung_HCA".Restzeit[14];
      JU    cR3V;

cR3R_2V:SET;
      S     #Belegt[18];
      L     "DB_Optimierung_HCA".Restzeit[8];
      T     "DB_Optimierung_HCA".Restzeit[18];
      JU    cR3V;

cR3V: A     #Belegt[11];
      A     #Lang[4];
      JC    cEnd;

      CALL  "FC_Optimierung_Pos"
      ( Pos        := 12,
        Umsetzzeit := #Umsetzzeit,
        Belegt     := #Belegt[12],
        Restzeit   := "DB_Optimierung_HCA".Restzeit[12]
      );

      AN    #Belegt[12];
      JC    cEnd;

      AN    #Belegt[2];
      AN    #Belegt[4];
      JC    cR3V_1R;

      AN    #Belegt[6];
      AN    #Belegt[4];
      JC    cR3V_1V;

      AN    #Belegt[14];
      AN    #Belegt[16];
      JC    cR3V_2R;

      AN    #Belegt[18];
      AN    #Belegt[16];
      JC    cR3V_2V;

      JU    cEnd;

cR3V_1R:SET;
      S     #Belegt[2];
      L     "DB_Optimierung_HCA".Restzeit[12];
      T     "DB_Optimierung_HCA".Restzeit[2];
      JU    cEnd;

cR3V_1V:SET;
      S     #Belegt[6];
      L     "DB_Optimierung_HCA".Restzeit[12];
      T     "DB_Optimierung_HCA".Restzeit[6];
      JU    cEnd;

cR3V_2R:SET;
      S     #Belegt[14];
      L     "DB_Optimierung_HCA".Restzeit[12];
      T     "DB_Optimierung_HCA".Restzeit[14];
      JU    cEnd;

cR3V_2V:SET;
      S     #Belegt[18];
      L     "DB_Optimierung_HCA".Restzeit[12];
      T     "DB_Optimierung_HCA".Restzeit[18];
      JU    cEnd;


cEnd: NOP   0;


NETWORK
TITLE = Auswertung Kurzware Links
//kurz Links
      L     "DB_Optimierung_HCA".Restzeit[1];
      L     "DB_Optimierung_HCA".Restzeit[5];
      >D;
      JC    kL1M;
      CAC;
kL1M: L     "DB_Optimierung_HCA".Restzeit[3];
      <D;
      JC    kL1;
      CAC;
kL1:  T     #Restzeit_Kurz_Links;

      L     "DB_Optimierung_HCA".Restzeit[13];
      L     "DB_Optimierung_HCA".Restzeit[17];
      >D;
      JC    kL2M;
      CAC;
kL2M: L     "DB_Optimierung_HCA".Restzeit[15];
      <D;
      JC    kL2;
      CAC;
kL2:  L     #Restzeit_Kurz_Links;
      >=D;
      JC    kLA;
      T     #Restzeit_Kurz_Links;

kLA:  L     #Restzeit_Kurz_Links;
      T     "DB_Optimierung_HCA".Restzeit_Kurz_Links;


NETWORK
TITLE = Auswertung Kurzware Rechts
//kurz Rechts
      L     "DB_Optimierung_HCA".Restzeit[2];
      L     "DB_Optimierung_HCA".Restzeit[6];
      >D;
      JC    kR1M;
      CAC;
kR1M: L     "DB_Optimierung_HCA".Restzeit[4];
      <D;
      JC    kR1;
      CAC;
kR1:  T     #Restzeit_Kurz_Rechts;

      L     "DB_Optimierung_HCA".Restzeit[14];
      L     "DB_Optimierung_HCA".Restzeit[18];
      >D;
      JC    kR2M;
      CAC;
kR2M: L     "DB_Optimierung_HCA".Restzeit[16];
      <D;
      JC    kR2;
      CAC;
kR2:  L     #Restzeit_Kurz_Rechts;
      >=D;
      JC    kRA;
      T     #Restzeit_Kurz_Rechts;

kRA:  L     #Restzeit_Kurz_Rechts;
      T     "DB_Optimierung_HCA".Restzeit_Kurz_Rechts;


NETWORK
TITLE = Auswertung Langware
//lang

      L     "DB_Optimierung_HCA".Restzeit[1];
      L     "DB_Optimierung_HCA".Restzeit[2];
      <D;
      JC    l_1V;
      CAC;

l_1V: T     #Restzeit_Lang;

      L     "DB_Optimierung_HCA".Restzeit[5];
      L     "DB_Optimierung_HCA".Restzeit[6];
      <D;
      JC    l_1R;
      CAC;

l_1R: L     #Restzeit_Lang;
      >=D;
      JC    l_1G;
      T     #Restzeit_Lang;

l_1G: L     "DB_Optimierung_HCA".Restzeit[3];
      L     "DB_Optimierung_HCA".Restzeit[4];
      <D;
      JC    l_1M;
      CAC;

l_1M: L     #Restzeit_Lang;
      <=D;
      JC    l_2;
      T     #Restzeit_Lang;

l_2:  L     "DB_Optimierung_HCA".Restzeit[13];
      L     "DB_Optimierung_HCA".Restzeit[14];
      <D;
      JC    l_2V;
      CAC;

l_2V: T     #Restzeit;

      L     "DB_Optimierung_HCA".Restzeit[17];
      L     "DB_Optimierung_HCA".Restzeit[18];
      <D;
      JC    l_2R;
      CAC;

l_2R: L     #Restzeit;
      >=D;
      JC    l_2G;
      T     #Restzeit;

l_2G: L     "DB_Optimierung_HCA".Restzeit[15];
      L     "DB_Optimierung_HCA".Restzeit[16];
      <D;
      JC    l_2M;
      CAC;

l_2M: L     #Restzeit;
      <=D;
      JC    l_AW;
      T     #Restzeit;

l_AW: L     #Restzeit_Lang;
      L     #Restzeit;
      >D;
      JC    l_TF;
      CAC;
l_TF: T     #Restzeit_Lang;
      T     "DB_Optimierung_HCA".Restzeit_Lang;


NETWORK
TITLE = Auswertung Großoptik Links
//gross links

      L     "DB_Optimierung_HCA".Restzeit[1];
      L     "DB_Optimierung_HCA".Restzeit[3];
      <D;
      JC    gL1V;
      CAC;
gL1V: L     "DB_Optimierung_HCA".Restzeit[5];
      <D;
      JC    gL1;
      CAC;
gL1:  T     #Restzeit_Gross_Links;

      L     "DB_Optimierung_HCA".Restzeit[13];
      L     "DB_Optimierung_HCA".Restzeit[15];
      <D;
      JC    gL2V;
      CAC;
gL2V: L     "DB_Optimierung_HCA".Restzeit[17];
      <D;
      JC    gL2;
      CAC;
gL2:  L     #Restzeit_Gross_Links;
      >D;
      JC    gLA;
      CAC;
      T     #Restzeit_Gross_Links;

gLA:  L     #Restzeit_Gross_Links;
      T     "DB_Optimierung_HCA".Restzeit_Gross_Links;


NETWORK
TITLE = Auswertung Großoptik Rechts
//gross rechts

      L     "DB_Optimierung_HCA".Restzeit[2];
      L     "DB_Optimierung_HCA".Restzeit[4];
      <D;
      JC    gR1V;
      CAC;
gR1V: L     "DB_Optimierung_HCA".Restzeit[6];
      <D;
      JC    gR1;
      CAC;
gR1:  T     #Restzeit_Gross_Rechts;

      L     "DB_Optimierung_HCA".Restzeit[14];
      L     "DB_Optimierung_HCA".Restzeit[16];
      <D;
      JC    gR2V;
      CAC;
gR2V: L     "DB_Optimierung_HCA".Restzeit[18];
      <D;
      JC    gR2;
      CAC;
gR2:  L     #Restzeit_Gross_Rechts;
      >D;
      JC    gRA;
      CAC;
      T     #Restzeit_Gross_Rechts;

gRA:  L     #Restzeit_Gross_Rechts;
      T     "DB_Optimierung_HCA".Restzeit_Gross_Rechts;

END_FUNCTION

FUNCTION "FC_Optimierung_Pos" : Void   // FC171, STL
{ S7_Optimized_Access := 'TRUE' }
// stored: AutoNumber false
   VAR_INPUT
      Pos : Int;
      Umsetzzeit : DInt;
   END_VAR
   VAR_OUTPUT
      Belegt : Bool;
   END_VAR
   VAR_IN_OUT
      Restzeit : DInt;
   END_VAR
   VAR_TEMP
      WT_DB : Int;
      Cmd : Int;
   END_VAR
BEGIN

NETWORK
TITLE = 
      L     0;
      T     #Restzeit;

      SET;
      R     #Belegt;

      L     0;
      L     "DB_POS".POS[#Pos].next_WT;
      ==I;
      BEC;
      S     #Belegt;
      +     100;
      T     #WT_DB;

      L     0;
      L     "DB_POS".POS[#Pos].WT_DB;
      ==I;
      L     "DB_POS".POS[#Pos].Soll_Expozeit;
      JC    setZ;
      L     "DB_POS".POS[#Pos].Restzeit;
setZ: T     #Restzeit;

      OPN   DB [#WT_DB];
      L     %DBW48;  //"DB_WT1".B_PNTER
retC: T     #Cmd;

      L     %DBW0;  //"DB_WT1".ANZAHL
      >=I;
      JC    ende;

      L     #Cmd;
      L     %DBW4;  //"DB_WT1".LENG
      *D;
      L     %DBW2;  //"DB_WT1".OFFSET
      +D;
      SLD   3;
      LAR1;

      L     #Restzeit;
      L     #Umsetzzeit;
      +D;
      T     #Restzeit;

      L     DBB [AR1, P#1.0];  //"DB_WT1".Befehl[#Cmd].Startpos
      L     18;
      >I;
      JC    ende;

      L     0;
      L     DBW [AR1, P#6.0];  //"DB_WT1".Befehl[#Cmd].Param_Ptr
      ==I;
      JC    nexC;
      SLD   3;
      LAR1;
      L     #Restzeit;
      L     DBD [AR1, P#0.0];
      +D;
      T     #Restzeit;

nexC: L     #Cmd;
      +     1;
      JU    retC;


ende: NOP   0;

END_FUNCTION

FUNCTION "FC_WT_MANAGER" : Void   // FC40, STL
TITLE = WT-Manager
{ S7_Optimized_Access := 'FALSE' }
AUTHOR : MS
// Verwaltung der Wt an Auf- und Ausgabestationen
// Technologiezuweisung
// stored: AutoNumber false
   VAR_TEMP
      FW_kommt : Bool;
      FW_in_Pos : Bool;
      Ziel_FW : Bool;
      STAND_POS : Byte;
      Param : DWord;
      AutoDelete : Bool;
      DeleteAll : Bool;
      Anforderung_QF : Bool;
      Sperre_TW : Bool;
   END_VAR
BEGIN

NETWORK
TITLE = Technologie
// Zuweisung on Technologien
//Programme laden

      CALL  "FC_Rez_to_DB45";

      CALL  "FC_AEND_WT";


NETWORK
TITLE = Check Querförderer
      A     "DI_QF_WR02_03".Zst.Req_WR02_In;
      O     "DI_QF_WR02_03".Zst.Req_WR03_In;
      O     "DI_QF_WR02_03".Zst.Req_WR02_Out;
      O     "DI_QF_WR02_03".Zst.Req_WR03_Out;
      O     "DI_QF_WR02_03".Out.WR02_einfahren;
      O     "DI_QF_WR02_03".Out.WR02_ausfahren;
      O     "DI_QF_WR02_03".Out.WR03_einfahren;
      O     "DI_QF_WR02_03".Out.WR03_ausfahren;
      =     #Anforderung_QF;

      A     "DI_QF_WR02_03".Zst.Req_WR02_In;
      O     "DI_QF_WR02_03".Zst.Req_WR03_In;
      O     "DI_QF_WR02_03".Zst.Req_WR02_Out;
      O     "DI_QF_WR02_03".Zst.Req_WR03_Out;
      A     "DI_QF_WR02_03".Zst.TW_sicher;
      O     "DI_QF_WR02_03".Out.WR02_einfahren;
      O     "DI_QF_WR02_03".Out.WR02_ausfahren;
      O     "DI_QF_WR02_03".Out.WR03_einfahren;
      O     "DI_QF_WR02_03".Out.WR03_ausfahren;
      =     #Sperre_TW;


NETWORK
TITLE = Beladestände
      A     "DB_ANLAGE".BA.Simulation;
      =     #AutoDelete;
      SET;
      =     #DeleteAll;

